INTERFACE I_PosMover

PROPERTY TargetPosition : LREAL
GET
END_GET
END_PROPERTY

END_INTERFACE

(* stored: Version 1.1.0.1
   Itf I_PosMover: Id {4bc065f6-a9ce-4bfb-b7d8-02f12e6af33f}
   Property TargetPosition: Id {4d48894c-81f1-496b-ae1d-9c595250bb94}
   Get Get: Id {17c9eee3-1f96-40d1-9334-cfdb6b9fbcae} *)
